// TwinCAT 3 PLC project Main
// Title: nepionic-cyclic
// Company: nepionic
// ProjectVersion: 0.1.0
// ProgramVersion: 3.1.4026.1+c9eadab3edd020c56c333d811d5b3c408c2550c8
// project tree:
//   / I_Cyclic.TcIO

// ---- I_Cyclic.TcIO
INTERFACE PUBLIC I_Cyclic EXTENDS __System.IQueryInterface

METHOD PUBLIC CyclicCall
END_METHOD

END_INTERFACE
